(* PLC project Unnamed, Unknown Unnamed 1 *)
(* stored: creationDateTime 2026-05-07T10:32:22, modificationDateTime 2026-05-07T10:32:22 *)

PROGRAM main
  VAR
    Timer_Pause : TON;
    Timer_Lys : TON;
    TimerLysOn : BOOL;
    PresetTime : TIME := T#500ms;
  END_VAR

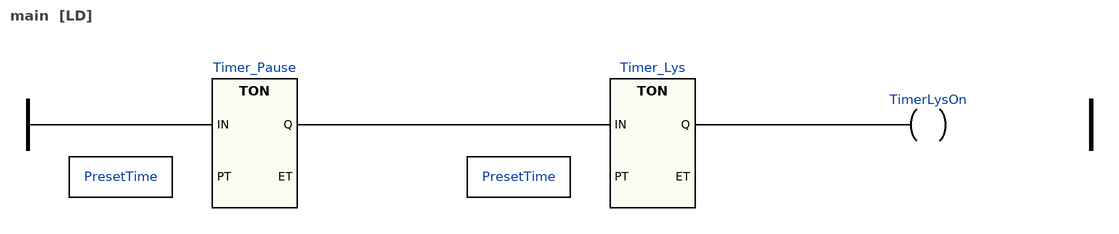
(* LD diagram, written out as Structured Text *)
Timer_Pause(IN := TRUE, PT := PresetTime);
Timer_Lys(IN := Timer_Pause.Q, PT := PresetTime);
TimerLysOn := Timer_Lys.Q;
END_PROGRAM

CONFIGURATION Config0
  RESOURCE Res0 ON PLC
    TASK task0(INTERVAL := T#20ms, PRIORITY := 1);
    PROGRAM instance0 WITH task0 : main;
  END_RESOURCE
END_CONFIGURATION
